# EPICS substitutions: iocBoot/ioc4idHHLM/substitutions/PI_E816.substitutions
file "$(MOTOR)/db/motor.db"
{
pattern
{N,  M,        DTYP,      C,  S,  DESC,          EGU,      DIR,  VELO,  VBAS,  ACCL,  BDST,  BVEL,  BACC,  MRES,   PREC,  DHLM,   DLLM,   INIT}
{4,  "m$(N)",  "PIE816",  0,  0,  "motor $(N)",  mm,       Pos,  1,     .1,    .2,    0,     1,      .2,   2.5e-4, 5,     100,    -100,   ""}
}
